Staubli VAL3: IN.pjx

--- IN.pjx ---
Parameters version=s7.5 stackSize=5000 millimeterUnit=true
Program file=find.pgx
Program file=get.pgx
Program file=getItem.pgx
Program file=getSize.pgx
Program file=getStatus.pgx
Program file=insert.pgx
Program file=isActive.pgx
Program file=isEnable.pgx
Program file=load.pgx
Program file=onEdit.pgx
Program file=onInsert.pgx
Program file=onProgEnd.pgx
Program file=onRun.pgx
Program file=onStart.pgx
Program file=onStop.pgx
Program file=reset.pgx
Program file=save.pgx
Program file=setActive.pgx
Program file=setEnable.pgx
Program file=setItem.pgx
Program file=stopRobot.pgx
Data file=IN.dtx
Library alias=saveInOut path=Disk://saveInputOutput/saveInputOutput.pjx
Library alias=use path=Disk://kernel/userPage/userPage.pjx
Library alias=language path=Disk://kernel/language/language.pjx
Library alias=cycleStatus path=Disk://cycleStatus/cycleStatus.pjx
Type name=dioItem path=Disk://kernel/template/dioItem/dioItem.pjx
Type name=aioItem path=Disk://kernel/template/aioItem/aioItem.pjx

--- find.pgx ---
public program find(string& x_sItem[], bool& x_bFound[])
  local num i
  local num l_nSize
  local string l_sItem
begin
  // find an item in the list
  x_bFound=isDefined(saveInOut:dInput[x_sItem])
end

--- get.pgx ---
public program get(string& x_sItem[], num x_nIndex)
  local num l_nSize
  local string l_sKey
  local num i
begin
  x_sItem=sKey[x_nIndex]

end

--- getItem.pgx ---
public program getItem(string& x_sItem, string& x_sId)
begin
  // get the name
  x_sItem=saveInOut:dInput[x_sId].sName
end

--- getSize.pgx ---
public program getSize(num& x_nSize[])
begin
  // size
  x_nSize=size(saveInOut:dInput)
end

--- getStatus.pgx ---
public program getStatus(bool& x_bStatus[], string x_sItem)
  local num l_nSize
begin
  // give back the status
  x_bStatus=saveInOut:dInput[x_sItem].dDio
end

--- insert.pgx ---
public program insert(string x_sItem, bool& x_bDone)
begin
  // insert a new item
  if isDefined(saveInOut:dInput[x_sItem])==false
    x_bDone=true
    insert(saveInOut:dInput[x_sItem])
  else
    // already exist
    x_bDone=false
  endIf

end

--- isActive.pgx ---
public program isActive(bool& x_bActive[], string x_sItem)
  local num l_nSize
begin
  // check if is active
  x_bActive=saveInOut:dInput[x_sItem].bActive
end

--- isEnable.pgx ---
public program isEnable(bool& x_bEnable[], string x_sItem)
  local num l_nSize
begin
  // check if is active
  x_bEnable=saveInOut:dInput[x_sItem].bEnable
end

--- onEdit.pgx ---
public program onEdit(string& x_sItem[])
  local string l_sItem[3]
  local num l_nCount
  local string l_sFlag[3]
  local string l_sName[3]
  local num i
  local string l_sData
  local num l_nFlag
  local string l_sMessage
  local num l_nNum
  local string l_sId
begin
  // show the real name
  l_sData=x_sItem
  do
    // sMode
    i=find(l_sData,"AND")
    if i!=-1
      i=i+len("AND")+1
    else
      i=find(l_sData,"OR")
      if i!=-1
        i=i+len("OR")+1
      endIf
    endIf
    //
    if i!=-1
      l_sItem[l_nCount]=left(l_sData,i)
      l_sData=right(l_sData,len(l_sData)-i)
    else
      l_sItem[l_nCount]=l_sData
    endIf
    l_nFlag=find(l_sItem[l_nCount],">")
    // l_bMode
    if find(l_sItem[l_nCount],">ON")!=-1
      l_sFlag[l_nCount]=">ON"+chr(10)
    else
      l_sFlag[l_nCount]=">OFF"+chr(10)
    endIf
    // sItem
    l_sItem[l_nCount]=left(l_sItem[l_nCount],l_nFlag)
    l_sId=l_sItem[l_nCount]
    l_sName[l_nCount]=saveInOut:dInput[l_sId].sName
    l_nCount=l_nCount+1
  until i==-1
  // show the ID+name
  l_sMessage=""
  for i=0 to 2
    if l_sItem[i]!=""
      l_sMessage=l_sMessage+l_sItem[i]+"["+l_sName[i]+"]"+l_sFlag[i]
    endIf
  endFor
  // popUp IT
  popUpMsg(l_sMessage)
end

--- onInsert.pgx ---
public program onInsert(string& x_sItem[])
  local num l_nSize
  local string l_sEvent
  local num i
  local num l_nKey
  local string l_sMessage
  local string l_sItem
  local string l_sOperator
  local bool l_bActive
  local num l_nIndex
  local string l_sItemList
  local num l_nSizeList
  local string l_sKey
  local string l_sName
begin
  x_sItem=""
  call getSize(l_nSizeList)
  do
    // create the list
    //
    call use:setSizeList(10,0,28,11)
    call use:listcreate("INPUT ")
    // start from the first
    l_sKey=first(saveInOut:dInput)
    while l_sKey!=""
      // scan
      call isActive(l_bActive,l_sKey)
      if l_bActive
        // insert into the list
        l_sName=saveInOut:dInput[l_sKey].sName
        l_sItemList=l_sKey+" {"+l_sName+"}"
        call use:listadd(l_sItemList)
      endIf
      // next
      l_sKey=next(saveInOut:dInput[l_sKey])
    endWhile
    //
    // display the list
    //
    call use:listredraw(min(l_nIndex-use:nView,0))
    //
    // wait a KEY
    //
    do
      l_nKey=get()
      // get one input from the list
      call use:listevent(l_nKey,l_nIndex,l_sEvent)
      if l_nKey==255
        return
      endIf
    until l_nKey==270
    //
    // insert the sentence
    //
    if l_sEvent==""
      return
    else
      l_sEvent=left(l_sEvent,find(l_sEvent,"{")-1)
    endIf
    l_sItem=l_sItem+l_sEvent
    // get the status ON-OFF
    call use:stringToArray("ON,OFF",sMessage)
    call language:message(l_sMessage,40)
    call use:questionDialog(l_sMessage,sMessage,i)
    if i==1
      l_sItem=l_sItem+">ON"
    else
      if i==2
        l_sItem=l_sItem+">OFF"
      else
        // escape
        return
      endIf
    endIf
    l_nSize=l_nSize+1
    if l_nSize!=3
      // define the operator
      if l_sOperator==""
        call use:stringToArray("OR,AND",sMessage)
      else
        call use:stringToArray(l_sOperator,sMessage)
      endIf
      call language:message(l_sMessage,41)
      call use:questionDialog(l_sMessage,sMessage,i)
      if i==-1
        // escape
        return
      else
        if i==1
          l_sItem=l_sItem+" "+sMessage+" "
          l_sOperator="OR"
        else
          if i==2
            l_sItem=l_sItem+" "+sMessage[1]+" "
            l_sOperator="AND"
          endIf
        endIf
      endIf
    endIf
  until i==0 or l_nSize==3
  x_sItem=l_sItem
end

--- onRun.pgx ---
public program onRun(string& x_sItem[])
  local bool l_bMode[3]
  local string l_sItem[3]
  local num l_nFlag
  local bool l_bActive
  local num l_nSize
  local num i
  local num j
  local string l_sName
  local string l_sMode
  local dio l_dDigital[3]
  local num l_nCount
  local string l_sId
begin
  //
  // find how many time and fill sItem and l_bMode
  //
  l_nCount=-1
  do
    l_nCount=l_nCount+1
    // l_sMode
    i=find(x_sItem,"AND")
    if i==-1
      i=find(x_sItem,"OR")
      if i!=-1
        l_sMode="OR"
        i=i+len("OR")+1
      endIf
    else
      l_sMode="AND"
      i=i+len("AND")+1
    endIf
    //
    if i!=-1
      l_sItem[l_nCount]=left(x_sItem,i)
      x_sItem=right(x_sItem,len(x_sItem)-i)
    else
      l_sItem[l_nCount]=x_sItem
    endIf
    l_nFlag=find(l_sItem[l_nCount],">")
    // l_bMode
    if find(l_sItem[l_nCount],">ON")!=-1
      l_bMode[l_nCount]=true
    else
      l_bMode[l_nCount]=false
    endIf
    //sItem
    l_sItem[l_nCount]=left(l_sItem[l_nCount],l_nFlag)
  until i==-1
  //
  //LINK IT
  //
  call getSize(l_nSize)
  // Link all
  for i=0 to l_nCount
    l_sId=l_sItem[i]
    dioLink(l_dDigital[i],saveInOut:dInput[l_sId].dDio)
  endFor
  // link the noLink
  for i=l_nCount to 2
    l_sId=l_sItem[i]=l_sItem[l_nCount]
    dioLink(l_dDigital[i],saveInOut:dInput[l_sId].dDio)
    l_bMode[i]=l_bMode[l_nCount]
  endFor
  //
  // DO IT
  //
  if l_sMode==""
    if !(l_dDigital[0]==l_bMode[0] or !saveInOut:dInput[l_sItem[0]].bEnable)
      call stopRobot()
      // wait the signal
      wait(l_dDigital[0]==l_bMode[0])
      cycleStatus:bWait=false
    endIf
  elseIf l_sMode=="OR"
    if !((l_dDigital[0]==l_bMode[0] or !saveInOut:dInput[l_sItem[0]].bEnable)or(l_dDigital[1]==l_bMode[1] or !saveInOut:dInput[l_sItem[1]].bEnable)or(l_dDigital[2]==l_bMode[2] or !saveInOut:dInput[l_sItem[2]].bEnable))
      // mutex the motion status
      call stopRobot()
      // wait the signal
      wait(l_dDigital[0]==l_bMode[0] or l_dDigital[1]==l_bMode[1] or l_dDigital[2]==l_bMode[2])
      cycleStatus:bWait=false
    endIf
  elseIf l_sMode=="AND"
    if !((l_dDigital[0]==l_bMode[0] or !saveInOut:dInput[l_sItem[0]].bEnable)and(l_dDigital[1]==l_bMode[1] or !saveInOut:dInput[l_sItem[1]].bEnable)and(l_dDigital[2]==l_bMode[2] or !saveInOut:dInput[l_sItem[2]].bEnable))
      // mutex the motion status
      call stopRobot()
      // wait the signal
      wait(l_dDigital[0]==l_bMode[0] and l_dDigital[1]==l_bMode[1] and l_dDigital[2]==l_bMode[2])
      cycleStatus:bWait=false
    endIf
  endIf
  //
end

--- onStart.pgx ---
public program onStart(string& x_sItem[])
// check and put all the boolean as the status of BIO-MIO-MODBUS-FIELDBUS-ARMIO
  local num i
  local num l_nModbusOut
  local num l_nFieldbusOut
  local bool l_bChange
  local num l_nResult
  local string l_sPath
  local bool l_bCheck
  local string l_sKey
begin
  if x_sItem=="init"
    //
    // DIGITAL INPUT
    //
    // set the default value
    call saveInOut:setInput(0)
//    // BIO
//    call saveInOut:setInput(1)
//    // BIO2 - MIO
//    call saveInOut:setInput(2)
//    // MODBUS
//    call saveInOut:setInput(3)
//    // USER
//    call saveInOut:setInput(4)
//    // REMIO
    //    call saveInOut:setInput(5)
    //.net
    call saveInOut:setInput(6)
    //
    // SAVE
    //
    call save(l_nResult)
    if l_nResult==0
      logMsg("[KERNEL] SUPERVISOR>Input: Save Done")
    else
      logMsg("error "+toString("",l_nResult)+" saving the saveInputInput")
      popUpMsg("error "+toString("",l_nResult)+" saving the saveInputInput")
    endIf
  endIf
  resize(sKey,1,1)
  sKey=""
  if isDefined(saveInOut:dInput["usrIn0"])
    append(sKey)
    sKey[0]="usrIn0"
  endIf
  if isDefined(saveInOut:dInput["usrIn1"])
    append(sKey)
    sKey[1]="usrIn1"
  endIf
  // insert the fIn or usrIn if exist
  if isDefined(saveInOut:dInput["fIn0"])
    sKey[2]="fIn0"
  endIf
  if isDefined(saveInOut:dInput["fIn1"])
    append(sKey)
    sKey[3]="fIn1"
  endIf
  l_sKey=first(saveInOut:dInput)
  i=size(sKey)-1
  //
  // copy all
  //
  while l_sKey!=""
    // use of number
    if find(l_sKey,"fIn")==-1 and find(l_sKey,"usrIn")==-1
      if !(sKey[0]=="" and i==0)
        append(sKey)
        i=i+1
      endIf
      sKey[i]=l_sKey
    endIf
    l_sKey=next(saveInOut:dInput[l_sKey])
  endWhile
end

--- reset.pgx ---
public program reset()
  local num l_nSize
  local num i
  local num l_nResult
  local string l_sKey
begin
  // reset it
  l_sKey="init"
  call onStart(l_sKey)
  // save it
  call save(l_nResult)
end

--- setActive.pgx ---
public program setActive(bool x_bActive, string x_sItem)
  local num l_nSize
begin
  // check if is active
  saveInOut:dInput[x_sItem].bActive=x_bActive
end

--- setEnable.pgx ---
public program setEnable(bool x_bEnable, string x_sItem)
  local num l_nSize
begin
  // check if is enable
  saveInOut:dInput[x_sItem].bEnable=x_bEnable
end

--- setItem.pgx ---
public program setItem(string x_sItem, string& x_sId[])
  local num l_nSize
begin
  // set the ITEM name
  saveInOut:dInput[x_sId].sName=x_sItem
end

--- stopRobot.pgx ---
program stopRobot()
begin
  // mutex the motion status
  setMutex(cycleStatus:bMotionToken)
  cycleStatus:bWait=true
  stopMove()
  // check that the robot has been stopped
  if watch(cycleStatus:bMoveStopped==true,10)==false
    popUpMsg("error stopping the robot using an INPUT ")
    logMsg("error stopping the robot using an INPUT ")
    wait(cycleStatus:bMoveStopped==true)
  endIf
end
